TYPE TcoSmartFunctionKitResponse_v_4_x_x : 
STRUCT
    AxisInReference : BOOL;
    ProgramActive : BOOL;
    LastPressingOk : BOOL;
    LastPressingNok : BOOL;
    SensorTared : BOOL;
    PressReady : BOOL;
    Error : BOOL;
    Warning : BOOL;
    RequestPossible : BOOL;
    ResponsAvialable : BOOL;
    NotificationAvailable : BOOL;
    EmergencyOffActive : BOOL;
    SafeStandstillActive : BOOL;
END_STRUCT
END_TYPE

(* stored: Version 1.1.0.1, ProductVersion 3.1.4024.11
   DUT TcoSmartFunctionKitResponse_v_4_x_x: Id {c056394b-7bb2-43c5-b5ef-f1b8ce1f9bca} *)
